FUNCTION_BLOCK CardboardEx EXTENDS SectionEx
VAR_IN_OUT
	benderLeft : FoldingMachine;
	
	robotLeft, robotRight : RobotA22;
	
	skidLeft, skidRight : SkidMagazine;
	magazineLeft, magazineRight : SkidMagazine;
	
	wrapper : WrapMachine;
	
	insertionLeft, insertionRight : Insertion;
	pistonBottom : SimplePiston;
	
	suctionTopLeft : ARRAY[*] OF SuctionPad; (*1..3*)
	suctionTopRight : ARRAY[*] OF SuctionPad; (*1..3*)
	suctionBottomLeft : ARRAY[*] OF SuctionPad; (*1..3*)
	suctionBottomRight : ARRAY[*] OF SuctionPad; (*1..3*)
	
	suctionBottom : ARRAY[*] OF SuctionPad; (*1..2*)
END_VAR
VAR	
	step : (IDLE, LOAD_SIDES_CORNERS, LOAD_TOP_BOTTOM, PUSH, TARGET_WRAP_POSITION, WRAP_AND_RELEASE, COMPLETE := 1050);
	
	masterLoadStep : INT;
	loadStepLeft, loadStepRight : INT;
	
	iWrap : INT;
	wrapPoints : INT;
	wrapRotations : INT;
	masterLength : INT;
	
	releaseDelayTimer : TON;
END_VAR
VAR //local types
	topLeftFoldsArr, topRightFoldsArr, bottomLeftFoldsArr, bottomRightFoldsArr : ARRAY[0..CONSTS.maxPairs] OF INT;
	
	//materialsArr : ARRAY[0..Consts.maxPairs] OF PositionMaterials;
	materialsArr : ARRAY[0..2*Consts.maxPairs] OF PositionMaterials;
	
	recipesCombined : BOOL;
	
	demoHeight : REAL := 640; //mm
	
	innerLoadedMaterials, outerLoadedMaterials : ARRAY[Surface.TOP..Surface.BOTTOM_RIGHT] OF STRING;
	//inner: cardboard by default
	//outer: corner guard by default
END_VAR
VAR CONSTANT
	releaseDelay : TIME := T#2000MS;
END_VAR
VAR
	//AOIs encapsulate functionality and reduce the number of module variables
	aoiCornerGuardLeft, aoiCornerGuardRight : AOI_LoadCornerGuard;
	aoiCornerCardboardLeft, aoiCornerCardboardRight : AOI_LoadCornerCardboard;
	aoiFlatCardboardLeft, aoiFlatCardboardRight : AOI_LoadFlatCardboard;
	
	//for testing only
	latchLeft, latchRight : BOOL; //prevents sliders from overshooting the inner limit sensor
	suctionEnableTopLeft, suctionEnableTopRight, suctionEnableBottomLeft, suctionEnableBottomRight : BOOL;
END_VAR

aoiBlocks();

SUPER^();

METHOD PROTECTED aoiBlocks : BOOL
VAR_INPUT
END_VAR
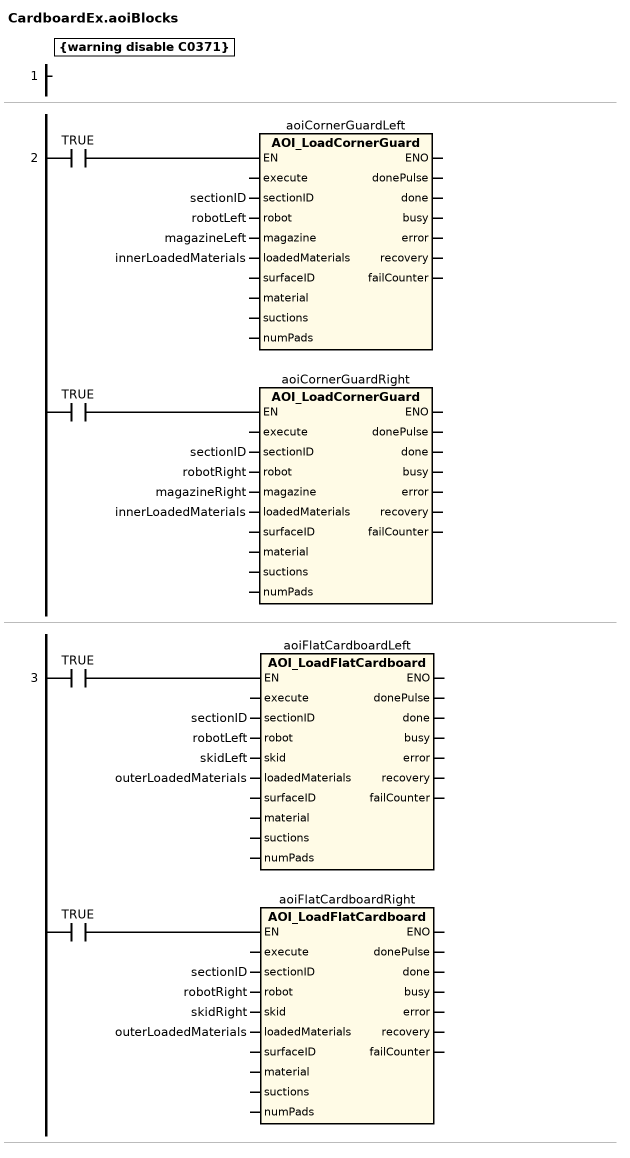
// NETWORK 1
// label: {warning disable C0371}

// NETWORK 2
aoiCornerGuardLeft(
    sectionID := sectionID,
    robot := robotLeft,
    magazine := magazineLeft,
    loadedMaterials := innerLoadedMaterials); // AOI_LoadCornerGuard
aoiCornerGuardRight(
    sectionID := sectionID,
    robot := robotRight,
    magazine := magazineRight,
    loadedMaterials := innerLoadedMaterials); // AOI_LoadCornerGuard

// NETWORK 3
aoiFlatCardboardLeft(
    sectionID := sectionID,
    robot := robotLeft,
    skid := skidLeft,
    loadedMaterials := outerLoadedMaterials); // AOI_LoadFlatCardboard
aoiFlatCardboardRight(
    sectionID := sectionID,
    robot := robotRight,
    skid := skidRight,
    loadedMaterials := outerLoadedMaterials); // AOI_LoadFlatCardboard
END_METHOD

METHOD PROTECTED combine : BOOL
VAR_IN_OUT
	cardboard : ARRAY[*] OF PositionMaterials;
	cornerGuard : ARRAY[*] OF PositionMaterials;
	
	combined : ARRAY[*] OF PositionMaterials;
END_VAR
VAR_INPUT
	cardboard_over_cornerGuard : BOOL;
END_VAR
VAR_INST
	topLength : REAL;
	leftLength : REAL;
	rightLength : REAL;
	bottomLength : REAL;
	
	topLeftLength : REAL;
	topRightLength : REAL;
	bottomLeftLength : REAL;
	bottomRightLength : REAL;
	
	outerMaterialLength : REAL;
	innerMaterialLength : REAL;
	
	i : INT;
	iCardboard : INT;
	iCornerGuard : INT;
END_VAR
FOR i:=0 TO CONSTS.maxPairs*2 BY 1 DO
	IF //no more cardboard (reached end of array or unused entries), 
		(iCardboard >= CONSTS.maxPairs OR_ELSE NOT PositionIsValid(cardboard[iCardboard])) AND_THEN //no more valid cardboard entries
		iCornerGuard < CONSTS.maxPairs AND_THEN //still has remaining corner guard
		PositionIsValid(cornerGuard[iCornerGuard]) //remaining corner guard is valid		
	THEN //finish with cornerguard
		combined[i] := cornerGuard[iCornerGuard];
		iCornerGuard := iCornerGuard + 1;
		CONTINUE;
	END_IF
	
	IF //no more cornerguard (reached end of array or unused entries)
		(iCornerGuard >= CONSTS.maxPairs OR_ELSE NOT PositionIsValid(cornerGuard[iCornerGuard])) AND_THEN
		iCardboard < CONSTS.maxPairs AND_THEN
		PositionIsValid(cardboard[iCardboard])
	THEN //finish with cardboard
		combined[i] := cardboard[iCardboard];
		iCardboard := iCardboard + 1;
		CONTINUE;
	END_IF
	
	(*
	IF NOT cardboard_over_cornerGuard THEN //cardboard on inside
		setOrder(cardboard, cornerGuard, combined, iCardboard, iCornerGuard, i);
		
	ELSE //cardboard on outside
		setOrder(cornerGuard, cardboard, combined, iCornerGuard, iCardboard, i);
		
	END_IF
	*)
END_FOR

combine := TRUE;
END_METHOD

METHOD PROTECTED load : BOOL
VAR_INPUT
	pairIndex : INT;
END_VAR
VAR_OUTPUT
	error : BOOL;
END_VAR
VAR
	pair : REFERENCE TO PositionMaterials REF= materialsArr[pairIndex];
	nextPair : REFERENCE TO PositionMaterials;
END_VAR
(*
unlike other sections, the load() function for cardboard + corner guard only loads the corners
to load flat cardboards, use the function loadFlats()
*)
{warning disable C0371}

IF robotLeft.error OR robotRight.error THEN
	RETURN;
ELSIF NOT (robotLeft.reserve(sectionID) AND robotRight.reserve(sectionID)) THEN //both robots must be reserved first
	RETURN;
END_IF

IF pairIndex + 1 < CONSTS.maxPairs THEN
	nextPair REF= materialsArr[pairIndex + 1];
END_IF

CASE masterLoadStep OF
	0: //check if next pair (which is to be placed over this pair) has the same position as this pair
		IF pairIndex + 1 >= CONSTS.maxPairs THEN //no next pair - NOTE: final pair is index 15 (16-1), not 16
			masterLoadStep := 10;
			loadStepLeft := loadStepRight := 0;
			
		ELSIF pair.position < nextPair.position THEN
			masterLoadStep := 10;
			loadStepLeft := loadStepRight := 0;
		(*	
		ELSIF MatchesMaterialType(pair:= nextPair, materialType:= 'CAR') AND_THEN loadCornerCardboards(pairIndex:= pairIndex + 1) THEN
			masterLoadStep := 10;
			loadStepLeft := loadStepRight := 0;
		*)
		ELSIF MatchesMaterialType(pair:= nextPair, materialPrefix:= 'COR') AND_THEN loadCornerGuards(pairIndex:= pairIndex + 1) THEN
			masterLoadStep := 10;
			loadStepLeft := loadStepRight := 0;
			
		END_IF
		
	10: //load this pair's side cardboards
		IF
			loadFlatCardboardsEx(
				robot:= robotLeft, 
				aoiLoad:= aoiFlatCardboardLeft, 
				loadStep:= loadStepLeft, 
				pairIndex:= pairIndex, 
				includeTop:= FALSE, 
				includeLeft:= TRUE, 
				includeRight:= FALSE, 
				includeBottom:= FALSE, 
				error=> )
			AND
			loadFlatCardboardsEx(
				robot:= robotLeft, 
				aoiLoad:= aoiFlatCardboardLeft, 
				loadStep:= loadStepLeft, 
				pairIndex:= pairIndex, 
				includeTop:= FALSE, 
				includeLeft:= FALSE, 
				includeRight:= TRUE, 
				includeBottom:= FALSE, 
				error=> )
		THEN
			masterLoadStep := 20;
			loadStepLeft := loadStepRight := 0;
		END_IF
		
	20: //load current pair
		IF
			MatchesMaterialType(pair:= pair, materialPrefix:= 'CAR') AND_THEN loadCornerCardboards(pairIndex:= iPair) OR_ELSE
			MatchesMaterialType(pair:= pair, materialPrefix:= 'COR') AND_THEN loadCornerGuards(pairIndex:= iPair)
		THEN //is cardboard
			loadStepLeft := loadStepRight := 0;
			masterLoadStep := COMPLETE;
		END_IF
	
	COMPLETE:
		robotLeft.release(sectionID);
		robotRight.release(sectionID);
		
		loadStepLeft := loadStepRight := 0;
		masterLoadStep := 0;
		load := TRUE;
	
END_CASE
END_METHOD

METHOD PROTECTED loadCornerCardboards : BOOL
VAR_INPUT
	pairIndex : INT;
END_VAR
VAR_OUTPUT
	error : BOOL;
END_VAR
VAR
	errorLeft, errorRight : BOOL;
	leftSuctionArr, rightSuctionArr : POINTER TO SuctionPad;
	leftNextSet, rightNextSet : INT;
	leftMaterial, rightMaterial : STRING;
	leftFold, rightFold : INT;
	
	pair : REFERENCE TO PositionMaterials REF= materialsArr[pairIndex];
	topLeftFold : INT := topLeftFoldsArr[pairIndex];
	topRightFold : INT := topRightFoldsArr[pairIndex];
	bottomLeftFold : INT := bottomLeftFoldsArr[pairIndex];
	bottomRightFold : INT := bottomRightFoldsArr[pairIndex];
END_VAR
{warning disable C0371}

loadCornerCardboards := 
	loadCornerCardboardsEx(
		robot:= robotLeft, 
		aoiLoad:= aoiCornerCardboardLeft, 
		loadStep:= loadStepLeft, 
		pairIndex:= pairIndex, 
		includeTopLeft:= TRUE, 
		includeTopRight:= FALSE, 
		includeBottomLeft:= TRUE, 
		includeBottomRight:= FALSE, 
		error=> errorLeft)
	AND
	loadCornerCardboardsEx(
		robot:= robotRight, 
		aoiLoad:= aoiCornerCardboardRight, 
		loadStep:= loadStepRight, 
		pairIndex:= pairIndex, 
		includeTopLeft:= FALSE, 
		includeTopRight:= TRUE, 
		includeBottomLeft:= FALSE, 
		includeBottomRight:= TRUE, 
		error=> errorLeft);
		
error := errorLeft OR errorRight;

(*
CASE cornerSetLeft OF
	0:
		leftNextSet := Surface.TOP_RIGHT;
		cornerSetLeft := 0;
		
	Surface.TOP_RIGHT: 
		leftNextSet := Surface.TOP_LEFT;
		leftSuctionArr := suctionTopRight;
		leftMaterial := pair.topRight;
		leftFold := topRightFold;
		
	Surface.TOP_LEFT: 
		leftNextSet := Surface.BOTTOM_RIGHT;
		leftSuctionArr := suctionTopLeft;
		leftMaterial := pair.topLeft;
		leftFold := topLeftFold;
		
	Surface.BOTTOM_RIGHT:
		leftNextSet := Surface.BOTTOM_LEFT;
		leftSuctionArr := suctionBottomRight;
		leftMaterial := pair.bottomRight;
		leftFold := bottomRightFold;
		
	Surface.BOTTOM_LEFT: 
		leftNextSet := COMPLETE;
		leftSuctionArr := suctionBottomLeft;
		leftMaterial := pair.bottomLeft;
		leftFold := bottomLeftFold;
END_CASE
IF
	(cornerSetLeft = 0 OR cornerSetLeft = COMPLETE) OR_ELSE
	leftCornerSequence(
		robot:= robotLeft, 
		skid:= skidLeft, 
		suctions := leftSuctionArr,
		loadStep:= loadStepLeft, 
		surfaceID:= cornerSetLeft,
		material:= pair.topRight, 
		foldPos0:= topRightFold, 
		foldPos1:= 0, 
		error=> )
THEN
	cornerSetLeft := leftNextSet;
	loadStepLeft := 0;
END_IF


CASE cornerSetRight OF
	0:
		cornerSetRight := Surface.TOP_RIGHT;
		rightSuctionArr := suctionTopRight;
		
	Surface.TOP_RIGHT:		
		rightNextSet := Surface.BOTTOM_RIGHT;
		rightSuctionArr := suctionTopRight;
		rightMaterial := pair.topRight;
		rightFold := topRightFold;
		
	Surface.BOTTOM_RIGHT: 
		rightNextSet := COMPLETE;
		rightSuctionArr := suctionBottomRight;
		rightMaterial := pair.bottomRight;
		rightFold := bottomRightFold;		
END_CASE
IF
	(cornerSetRight = 0 OR cornerSetRight = COMPLETE) OR_ELSE
	rightCornerSequence(
		robot:= robotRight, 
		skid:= skidRight, 
		suctions := rightSuctionArr,
		loadStep:= loadStepRight, 
		material:= pair.topRight, 
		surfaceID:= cornerSetRight,
		foldPos0:= pair.topRightFold, 
		foldPos1:= 0, 
		error=> )
THEN
	cornerSetRight := rightNextSet;
	loadStepRight := 0;
END_IF



IF cornerSetLeft = COMPLETE AND cornerSetRight = COMPLETE THEN
	loadCornerCardboards := TRUE;
	
	loadStepLeft := loadStepRight := 0;
	cornerSetLeft := cornerSetRight := 0;
END_IF
*)
END_METHOD

METHOD PROTECTED loadCornerCardboardsEx : BOOL
VAR_IN_OUT
	robot : RobotA22;
	aoiLoad : AOI_LoadCornerCardboard;
	loadStep : INT;
END_VAR
VAR_INPUT
	pairIndex : INT;
	includeTopLeft, includeTopRight, includeBottomLeft, includeBottomRight : BOOL;
END_VAR
VAR_OUTPUT
	error : BOOL;
END_VAR
VAR
	suctionsArrLeft, suctionsArrRight : POINTER TO SuctionPad;
	nextSetLeft, nextSetRight : INT;

	pair : REFERENCE TO PositionMaterials REF= materialsArr[pairIndex];
	topLeftFold : INT := topLeftFoldsArr[pairIndex];
	topRightFold : INT := topRightFoldsArr[pairIndex];
	bottomLeftFold : INT := bottomLeftFoldsArr[pairIndex];
	bottomRightFold : INT := bottomRightFoldsArr[pairIndex];
END_VAR
{warning disable C0371}

IF robot.error THEN
	error := TRUE;
	RETURN;
ELSIF robot.reservation <> sectionID AND_THEN NOT robot.reserve(sectionID) THEN
	RETURN;
ELSIF robot.tool <> sectionID AND_THEN NOT robot.changeEOAT(targetTool := sectionID) THEN
	RETURN;
END_IF

error := aoiLoad.error;

CASE loadStep OF
	0:
		loadStep := Surface.BOTTOM_LEFT;
		
	Surface.BOTTOM_LEFT:
		IF NOT includeBottomLeft OR aoiLoad.donePulse THEN
			aoiLoad.execute := FALSE;
			aoiLoad.material := '';
			loadStep := Surface.BOTTOM_RIGHT;
			RETURN;
		END_IF
		
		aoiLoad.surfaceID := loadStep;
		aoiLoad.material := pair.bottomLeft;
		aoiLoad.suctions := suctionBottomLeft;
		aoiLoad.numPads := UPPER_BOUND(suctionBottomLeft, 1) - LOWER_BOUND(suctionBottomLeft, 1) + 1;
		
		aoiLoad.foldPos0 := bottomLeftFold;
		aoiLoad.foldPos1 := 0;
		
		aoiLoad.execute := NOT aoiLoad.busy;
		
	Surface.BOTTOM_RIGHT:
		IF NOT includeBottomRight OR aoiLoad.donePulse THEN
			aoiLoad.execute := FALSE;
			aoiLoad.material := '';
			loadStep := Surface.TOP_LEFT;
			RETURN;
		END_IF
		
		aoiLoad.surfaceID := loadStep;
		aoiLoad.material := pair.bottomRight;
		aoiLoad.suctions := suctionBottomRight;
		aoiLoad.numPads := UPPER_BOUND(suctionBottomRight, 1) - LOWER_BOUND(suctionBottomRight, 1) + 1;
		
		aoiLoad.foldPos0 := bottomRightFold;
		aoiLoad.foldPos1 := 0;
		
		aoiLoad.execute := NOT aoiLoad.busy;
	
	Surface.TOP_LEFT:		
		IF NOT includeTopLeft OR aoiLoad.donePulse THEN
			aoiLoad.execute := FALSE;
			aoiLoad.material := '';
			loadStep := Surface.TOP_RIGHT;
			RETURN;
		END_IF
		
		aoiLoad.surfaceID := loadStep;
		aoiLoad.material := pair.top;
		aoiLoad.suctions := suctionTopLeft;
		aoiLoad.numPads := UPPER_BOUND(suctionTopLeft, 1) - LOWER_BOUND(suctionTopLeft, 1) + 1;
		
		aoiLoad.foldPos0 := topLeftFold;
		aoiLoad.foldPos1 := 0;
		
		aoiLoad.execute := NOT aoiLoad.busy;
		
	Surface.TOP_RIGHT:
		IF NOT includeTopRight OR aoiLoad.donePulse THEN
			aoiLoad.execute := FALSE;
			aoiLoad.material := '';
			loadStep := COMPLETE;
			RETURN;
		END_IF
		
		aoiLoad.surfaceID := loadStep;
		aoiLoad.material := pair.topRight;
		aoiLoad.suctions := suctionTopRight;
		aoiLoad.numPads := UPPER_BOUND(suctionTopRight, 1) - LOWER_BOUND(suctionTopRight, 1) + 1;
		
		aoiLoad.foldPos0 := topRightFold;
		aoiLoad.foldPos1 := 0;
		
		aoiLoad.execute := NOT aoiLoad.busy;
		
	COMPLETE:				
		robot.release(sectionID);
		
		aoiLoad.material := '';
		aoiLoad.execute := FALSE;
		
		loadCornerCardboardsEx := TRUE;
END_CASE
END_METHOD

METHOD loadCornerGuards : BOOL
VAR_INPUT
	pairIndex : INT;
END_VAR
VAR_OUTPUT
	error : BOOL;
END_VAR
VAR
	pair : REFERENCE TO PositionMaterials REF= materialsArr[pairIndex];
	errorLeft, errorRight : BOOL;
END_VAR
{warning disable C0371}

loadCornerGuards := 
	loadCornerGuardsEx(
		robot:= robotLeft, 
		aoiLoad:= aoiCornerGuardLeft, 
		loadStep:= loadStepLeft, 
		pairIndex:= pairIndex, 
		includeTopLeft:= TRUE, 
		includeTopRight:= FALSE, 
		includeBottomLeft:= TRUE, 
		includeBottomRight:= FALSE, 
		error=> errorLeft) 
	AND
	loadCornerGuardsEx(
		robot:= robotRight, 
		aoiLoad:= aoiCornerGuardRight, 
		loadStep:= loadStepRight, 
		pairIndex:= pairIndex, 
		includeTopLeft:= FALSE, 
		includeTopRight:= TRUE, 
		includeBottomLeft:= FALSE, 
		includeBottomRight:= TRUE, 
		error=> errorRight);
		
error := errorLeft OR errorRight;

(*
IF robotLeft.error OR robotRight.error THEN
	error := TRUE;
	RETURN;
	
ELSIF 
	(robotLeft.reservation <> sectionID AND_THEN NOT robotLeft.reserve(sectionID)) OR 
	(robotRight.reservation <> sectionID AND_THEN NOT robotRight.reserve(sectionID))
THEN //loading requires both robots be reserved together
	RETURN;
	
ELSIF //robots have wrong tool
	(robotLeft.tool <> sectionID AND_THEN NOT robotLeft.changeEOAT(targetTool := sectionID)) OR
	(robotRight.tool <> sectionID AND_THEN NOT robotRight.changeEOAT(targetTool := sectionID))
THEN
	RETURN;
	
END_IF

CASE loadStep OF
	0: //top and bottom
		IF aoiCornerGuardLeft.done AND aoiCornerGuardRight.done THEN
			aoiCornerGuardLeft.execute := aoiCornerGuardRight.execute := FALSE;
			aoiCornerGuardLeft.material := aoiCornerGuardRight.material := '';
			loadStep := 10;
			RETURN;
		END_IF
		
		aoiCornerGuardLeft.suctions := 0;
		aoiCornerGuardLeft.surfaceID := Surface.TOP;
		aoiCornerGuardLeft.material := pair.top;
		aoiCornerGuardLeft.numPads := 0;
		
		aoiCornerGuardRight.suctions := suctionBottom;
		aoiCornerGuardRight.surfaceID := Surface.BOTTOM;
		aoiCornerGuardRight.material := pair.bottom;
		aoiCornerGuardRight.numPads := 0;
		
		aoiCornerGuardLeft.execute := NOT aoiCornerGuardLeft.done AND NOT aoiCornerGuardLeft.busy;
		aoiCornerGuardRight.execute := NOT aoiCornerGuardRight.done AND NOT aoiCornerGuardRight.busy;
		
	10: //sides
		IF aoiCornerGuardLeft.done AND aoiCornerGuardRight.done THEN
			aoiCornerGuardLeft.execute := aoiCornerGuardRight.execute := FALSE;
			aoiCornerGuardLeft.material := aoiCornerGuardRight.material := '';
			loadStep := 10;
			RETURN;
		END_IF
		
		aoiCornerGuardLeft.suctions := 0;
		aoiCornerGuardLeft.surfaceID := Surface.LEFT;
		aoiCornerGuardLeft.material := pair.left;
		aoiCornerGuardLeft.numPads := 0;
		
		aoiCornerGuardRight.suctions := 0;
		aoiCornerGuardRight.surfaceID := Surface.RIGHT;
		aoiCornerGuardRight.material := pair.right;
		aoiCornerGuardRight.numPads := 0;
		
		aoiCornerGuardLeft.execute := NOT aoiCornerGuardLeft.done AND NOT aoiCornerGuardLeft.busy;
		aoiCornerGuardRight.execute := NOT aoiCornerGuardRight.done AND NOT aoiCornerGuardRight.busy;
		
	COMPLETE:
		loadStep := 0;
		loadCornerGuards := TRUE;
END_CASE

error := aoiCornerGuardLeft.error OR aoiCornerGuardRight.error;
*)
END_METHOD

METHOD loadCornerGuardsEx : BOOL
VAR_IN_OUT
	robot : RobotA22;
	aoiLoad : AOI_LoadCornerGuard;
	loadStep : INT;
END_VAR
VAR_INPUT
	pairIndex : INT;
	includeTopLeft, includeTopRight, includeBottomLeft, includeBottomRight : BOOL;
END_VAR
VAR_OUTPUT
	error : BOOL;
END_VAR
VAR
	pair : REFERENCE TO PositionMaterials REF= materialsArr[pairIndex];
END_VAR
{warning disable C0371}
IF robot.error THEN
	error := TRUE;
	RETURN;
ELSIF robot.reservation <> sectionID AND_THEN NOT robot.reserve(sectionID) THEN
	RETURN;
ELSIF robot.tool <> sectionID AND_THEN NOT robot.changeEOAT(targetTool := sectionID) THEN
	RETURN;
END_IF

error := aoiLoad.error;

CASE loadStep OF
	0:
		loadStep := Surface.BOTTOM_LEFT;
		
	Surface.BOTTOM_LEFT:
		IF NOT includeBottomLeft OR aoiLoad.donePulse THEN
			aoiLoad.execute := FALSE;
			aoiLoad.material := '';
			loadStep := Surface.BOTTOM_RIGHT;
			RETURN;
		END_IF
		
		aoiLoad.surfaceID := loadStep;
		aoiLoad.material := pair.bottomLeft;
		aoiLoad.suctions := suctionBottomLeft;
		aoiLoad.numPads := UPPER_BOUND(suctionBottomLeft, 1) - LOWER_BOUND(suctionBottomLeft, 1) + 1;
		
		aoiLoad.execute := NOT aoiLoad.busy;
		
	Surface.BOTTOM_RIGHT:
		IF NOT includeBottomRight OR aoiLoad.donePulse THEN
			aoiLoad.execute := FALSE;
			aoiLoad.material := '';
			loadStep := Surface.TOP_LEFT;
			RETURN;
		END_IF
		
		aoiLoad.surfaceID := loadStep;
		aoiLoad.material := pair.bottomRight;
		aoiLoad.suctions := suctionBottomRight;
		aoiLoad.numPads := UPPER_BOUND(suctionBottomRight, 1) - LOWER_BOUND(suctionBottomRight, 1) + 1;
		
		aoiLoad.execute := NOT aoiLoad.busy;
	
	Surface.TOP_LEFT:		
		IF NOT includeTopLeft OR aoiLoad.donePulse THEN
			aoiLoad.execute := FALSE;
			aoiLoad.material := '';
			loadStep := Surface.TOP_RIGHT;
			RETURN;
		END_IF
		
		aoiLoad.surfaceID := loadStep;
		aoiLoad.material := pair.top;
		aoiLoad.suctions := suctionTopLeft;
		aoiLoad.numPads := UPPER_BOUND(suctionTopLeft, 1) - LOWER_BOUND(suctionTopLeft, 1) + 1;
		
		aoiLoad.execute := NOT aoiLoad.busy;
		
	Surface.TOP_RIGHT:
		IF NOT includeTopRight OR aoiLoad.donePulse THEN
			aoiLoad.execute := FALSE;
			aoiLoad.material := '';
			loadStep := COMPLETE;
			RETURN;
		END_IF
		
		aoiLoad.surfaceID := loadStep;
		aoiLoad.material := pair.topRight;
		aoiLoad.suctions := suctionTopRight;
		aoiLoad.numPads := UPPER_BOUND(suctionTopRight, 1) - LOWER_BOUND(suctionTopRight, 1) + 1;
		
		aoiLoad.execute := NOT aoiLoad.busy;
		
	COMPLETE:				
		robot.release(sectionID);
		
		aoiLoad.material := '';
		aoiLoad.execute := FALSE;
		
		loadCornerGuardsEx := TRUE;
END_CASE
END_METHOD

METHOD PROTECTED loadFlatCardboards : BOOL
VAR_INPUT
	pairIndex : INT;
END_VAR
VAR_OUTPUT
	error : BOOL;
END_VAR
VAR
	pair : REFERENCE TO PositionMaterials REF= materialsArr[pairIndex];
	errorLeft, errorRight : BOOL;
END_VAR
{warning disable C0371}

loadFlatCardboards := 
	loadFlatCardboardsEx(
		robot:= robotLeft, 
		aoiLoad:= aoiFlatCardboardLeft, 
		loadStep:= loadStepLeft, 
		pairIndex:= pairIndex, 
		includeTop:= TRUE, 
		includeLeft:= FALSE, //left already loaded before
		includeRight:= FALSE, 
		includeBottom:= FALSE, 
		error=> errorLeft)
	AND
	loadFlatCardboardsEx(
		robot:= robotRight, 
		aoiLoad:= aoiFlatCardboardRight, 
		loadStep:= loadStepRight, 
		pairIndex:= pairIndex, 
		includeTop:= FALSE, 
		includeLeft:= FALSE, 
		includeRight:= FALSE, //right already loaded before
		includeBottom:= TRUE, 
		error=> errorRight);
		
error := errorLeft OR errorRight;

(*
IF robotLeft.error OR robotRight.error THEN
	error := TRUE;
	RETURN;
	
ELSIF 
	(robotLeft.reservation <> sectionID AND_THEN NOT robotLeft.reserve(sectionID)) OR 
	(robotRight.reservation <> sectionID AND_THEN NOT robotRight.reserve(sectionID))
THEN //loading requires both robots be reserved together
	RETURN;
	
ELSIF //robots have wrong tool
	(robotLeft.tool <> sectionID AND_THEN NOT robotLeft.changeEOAT(targetTool := sectionID)) OR
	(robotRight.tool <> sectionID AND_THEN NOT robotRight.changeEOAT(targetTool := sectionID))
THEN
	RETURN;
	
END_IF

CASE loadStep OF
	0: //top and bottom
		IF aoiFlatCardboardLeft.done AND aoiFlatCardboardRight.done THEN
			aoiFlatCardboardLeft.execute := aoiFlatCardboardRight.execute := FALSE;
			aoiFlatCardboardLeft.material := aoiFlatCardboardRight.material := '';
			loadStep := 10;
			RETURN;
		END_IF
		
		aoiFlatCardboardLeft.suctions := 0;
		aoiFlatCardboardLeft.surfaceID := Surface.TOP;
		aoiFlatCardboardLeft.material := pair.top;
		aoiFlatCardboardLeft.numPads := 0;
		
		aoiFlatCardboardRight.suctions := suctionBottom;
		aoiFlatCardboardRight.surfaceID := Surface.BOTTOM;
		aoiFlatCardboardRight.material := pair.bottom;
		aoiFlatCardboardRight.numPads := 0;
		
		aoiFlatCardboardLeft.execute := NOT aoiFlatCardboardLeft.done AND NOT aoiFlatCardboardLeft.busy;
		aoiFlatCardboardRight.execute := NOT aoiFlatCardboardRight.done AND NOT aoiFlatCardboardRight.busy;
		
	10: //sides
		IF aoiFlatCardboardLeft.done AND aoiFlatCardboardRight.done THEN
			aoiFlatCardboardLeft.execute := aoiFlatCardboardRight.execute := FALSE;
			aoiFlatCardboardLeft.material := aoiFlatCardboardRight.material := '';
			loadStep := 10;
			RETURN;
		END_IF
		
		aoiFlatCardboardLeft.suctions := 0;
		aoiFlatCardboardLeft.surfaceID := Surface.LEFT;
		aoiFlatCardboardLeft.material := pair.left;
		aoiFlatCardboardLeft.numPads := 0;
		
		aoiFlatCardboardRight.suctions := 0;
		aoiFlatCardboardRight.surfaceID := Surface.RIGHT;
		aoiFlatCardboardRight.material := pair.right;
		aoiFlatCardboardRight.numPads := 0;
		
		aoiFlatCardboardLeft.execute := NOT aoiFlatCardboardLeft.done AND NOT aoiFlatCardboardLeft.busy;
		aoiFlatCardboardRight.execute := NOT aoiFlatCardboardRight.done AND NOT aoiFlatCardboardRight.busy;
		
	COMPLETE:
		loadStepLeft := loadStepRight := 0;
		loadStep := 0;
		
		loadFlatCardboards := TRUE;
END_CASE

error := aoiFlatCardboardLeft.error OR aoiFlatCardboardRight.error;
*)
END_METHOD

METHOD loadFlatCardboardsEx : BOOL
VAR_IN_OUT
	robot : RobotA22;
	aoiLoad : AOI_LoadFlatCardboard;
	loadStep : INT;
END_VAR
VAR_INPUT
	pairIndex : INT;
	includeTop, includeLeft, includeRight, includeBottom : BOOL;
END_VAR
VAR_OUTPUT
	error : BOOL;
END_VAR
VAR
	pair : REFERENCE TO PositionMaterials REF= materialsArr[pairIndex];
END_VAR
IF robot.error THEN
	error := TRUE;
	RETURN;
ELSIF robot.reservation <> sectionID AND_THEN NOT robot.reserve(sectionID) THEN
	RETURN;
ELSIF robot.tool <> sectionID AND_THEN NOT robot.changeEOAT(targetTool := sectionID) THEN
	RETURN;
END_IF

error := aoiLoad.error;

CASE loadStep OF
	0:
		loadStep := Surface.TOP;
	
	Surface.TOP:	
		IF NOT includeTop OR aoiLoad.donePulse THEN
			aoiLoad.execute := FALSE;
			aoiLoad.material := '';
			loadStep := Surface.BOTTOM;
			RETURN;
		END_IF
		
		aoiLoad.surfaceID := Surface.TOP;
		aoiLoad.material := pair.top;
		aoiLoad.suctions := 0;
		aoiLoad.numPads := 0;
		
		aoiLoad.execute := NOT aoiLoad.busy;
		
	Surface.BOTTOM:
		IF NOT includeBottom OR aoiLoad.donePulse THEN
			aoiLoad.execute := FALSE;
			aoiLoad.material := '';
			loadStep := Surface.LEFT;
			RETURN;
		END_IF
		
		aoiLoad.surfaceID := Surface.BOTTOM;
		aoiLoad.material := pair.bottom;
		aoiLoad.suctions := suctionBottom;
		aoiLoad.numPads := UPPER_BOUND(suctionBottom, 1) - LOWER_BOUND(suctionBottom, 1) + 1;
		
		aoiLoad.execute := NOT aoiLoad.busy;
		
	Surface.LEFT:
		IF NOT includeLeft OR aoiLoad.donePulse THEN
			aoiLoad.execute := FALSE;
			aoiLoad.material := '';
			loadStep := Surface.RIGHT;
			RETURN;
		END_IF
		
		aoiLoad.surfaceID := Surface.LEFT;
		aoiLoad.material := pair.left;
		aoiLoad.suctions := 0;
		aoiLoad.numPads := 0;
		
		aoiLoad.execute := NOT aoiLoad.busy;
		
	Surface.RIGHT:
		IF NOT includeRight OR aoiLoad.donePulse THEN
			aoiLoad.execute := FALSE;
			aoiLoad.material := '';
			loadStep := COMPLETE;
			RETURN;
		END_IF
		
		aoiLoad.surfaceID := Surface.RIGHT;
		aoiLoad.material := pair.right;
		aoiLoad.suctions := 0;
		aoiLoad.numPads := 0;
		
		aoiLoad.execute := NOT aoiLoad.busy;
		
	COMPLETE:				
		robot.release(sectionID);
		
		aoiLoad.material := '';
		aoiLoad.execute := FALSE;
		
		loadFlatCardboardsEx := TRUE;
END_CASE
END_METHOD

METHOD PROTECTED maintenance : BOOL
VAR_INPUT
END_VAR
{warning disable C0371}
IF robotLeft.Done THEN
	robotLeft.clearCommand();
END_IF

IF robotRight.Done THEN
	robotRight.clearCommand();
END_IF
END_METHOD

METHOD PROTECTED manual : BOOL
VAR_INPUT
END_VAR
END_METHOD

METHOD PROTECTED process : BOOL
VAR_INPUT
	auto : BOOL;
END_VAR
VAR_OUTPUT
	error : BOOL;
END_VAR
VAR
	currentPair : REFERENCE TO PositionMaterials REF= materialsArr[iPair];
END_VAR
{warning disable C0371}

IF iPair >= CONSTS.maxPairs THEN
	process := TRUE;
	RETURN;
ELSIF NOT PositionIsValid(pair := currentPair) THEN
	iPair := iPair + 1;
	RETURN;
END_IF
(*
corrected sequence:
	load sides
	load corners
	load bottom
	load top
*)

CASE step OF
	IDLE:
		IF trigger.Q THEN
			step := LOAD_SIDES_CORNERS;
		END_IF
	
	LOAD_SIDES_CORNERS: //load
		IF
			(auto AND done) OR
			(NOT auto AND trigger.Q)
		THEN
			aoiCornerCardboardLeft.reset();
			aoiCornerCardboardRight.reset();
			
			aoiCornerGuardLeft.reset();
			aoiCornerGuardRight.reset();
			
			aoiFlatCardboardLeft.reset();
			aoiFlatCardboardRight.reset();
			
			step := LOAD_TOP_BOTTOM;
			RETURN;
		END_IF
		
		IF NOT done THEN
			done := load(pairIndex := iPair);
		END_IF
		
	LOAD_TOP_BOTTOM:
		IF
			(auto AND done) OR
			(NOT auto AND trigger.Q)
		THEN
			aoiCornerCardboardLeft.reset();
			aoiCornerCardboardRight.reset();
			
			aoiCornerGuardLeft.reset();
			aoiCornerGuardRight.reset();
			
			aoiFlatCardboardLeft.reset();
			aoiFlatCardboardRight.reset();
			
			step := PUSH;
			RETURN;
		END_IF
		
		IF NOT done THEN
			done := loadFlatCardboards(pairIndex := iPair);
		END_IF
		
	PUSH:
		IF
			(auto AND latchLeft AND latchRight AND pistonBottom.extended) OR
			(NOT auto AND trigger.Q)
		THEN
			step := TARGET_WRAP_POSITION;
			RETURN;
		END_IF
		
		insertionLeft.align(demoHeight+5);
		insertionRight.align(demoHeight+5);
		
		IF //align slider to 5mm gap above bundle height
			insertionLeft.sliderPos <> demoHeight+5 OR
			insertionRight.sliderPos <> demoHeight+5
		THEN
			RETURN;
		END_IF
		
		IF NOT latchLeft THEN
			latchLeft := insertionLeft.contact;
			insertionLeft.press();
		END_IF
		
		IF NOT latchRight THEN
			latchRight := insertionRight.contact;
			insertionRight.press();
		END_IF
		
		pistonBottom.extend();
		
	TARGET_WRAP_POSITION:		
		IF iWrap >= wrapPoints THEN
			step := COMPLETE;
			RETURN;
		END_IF
		
		IF materialsArr[iPair].position = materialsArr[iPair + 1].position THEN //if this and the next pair were loaded together
			masterLength := TO_INT( MAX( GetPairMasterLength(materialsArr[iPair]), GetPairMasterLength(materialsArr[iPair + 1]) ) );
			wrapPoints := MAX( materialsArr[iPair].wrapPoints, materialsArr[iPair + 1].wrapPoints );
			wrapRotations := MAX( materialsArr[iPair].wrapRotations, materialsArr[iPair + 1].wrapRotations );
		ELSE
			masterLength := TO_INT( GetPairMasterLength(materialsArr[iPair]) );
			wrapPoints := materialsArr[iPair].wrapPoints;
			wrapRotations := materialsArr[iPair].wrapRotations;
		END_IF
		
		(*
		directionCheckAndSet(
			wrapConveyorPos,
			(currentPair.position - masterLength/2) + (masterLength/(currentPair.wrapPoints + 1) * (iWrap + 1)));
		*)
		step := WRAP_AND_RELEASE;
		
	WRAP_AND_RELEASE:
		releaseDelayTimer(IN:= , PT:= releaseDelay, Q=> , ET=> );
		
		IF wrapper.ready THEN
			wrapper.wrap(wrapRotations);
			releaseDelayTimer.IN := TRUE;
		END_IF
		
		IF releaseDelayTimer.Q THEN
			SetSuctions(suctions := suctionTopLeft, state := FALSE);
			SetSuctions(suctions := suctionTopRight, state := FALSE);
			SetSuctions(suctions := suctionBottomLeft, state := FALSE);
			SetSuctions(suctions := suctionBottomRight, state := FALSE);
			
			insertionLeft.toHome();
			insertionRight.toHome();
			pistonBottom.retract();
		END_IF
		
		IF wrapper.done AND insertionLeft.home AND insertionRight.home AND pistonBottom.retracted THEN
			releaseDelayTimer.IN := FALSE;
			step := WRAP_AND_RELEASE;
		END_IF
	
	COMPLETE:
		iPair := iPair + 1;
		iWrap := wrapPoints := wrapRotations := 0;
		step := IDLE;
		
END_CASE
END_METHOD

METHOD PROTECTED ps_AbortCondition : BOOL
VAR_INPUT
END_VAR
{warning disable C0371}
ps_AbortCondition :=
	insertionLeft.error OR 
	insertionRight.error OR 
	robotLeft.error OR 
	robotRight.error OR
	wrapper.error;
END_METHOD

METHOD PROTECTED ps_Aborted : BOOL
VAR_INPUT
END_VAR
ps_Aborted := TRUE;
END_METHOD

METHOD PROTECTED ps_Aborting : BOOL
VAR_INPUT
END_VAR
{warning disable C0371}
insertionLeft.stop();
insertionRight.stop();
pistonBottom.stop();

aoiFlatCardboardLeft.reset();
aoiFlatCardboardRight.reset();

aoiCornerCardboardLeft.reset();
aoiCornerCardboardRight.reset();

aoiCornerGuardLeft.reset();
aoiCornerGuardRight.reset();

robotLeft.clearCommand();
robotRight.clearCommand();

//stop conveyors

ps_Aborting :=
	NOT insertionLeft.active AND
	NOT insertionRight.active AND
	NOT pistonBottom.busy AND
	NOT robotLeft.Busy AND
	NOT robotRight.Busy;
END_METHOD

METHOD PROTECTED ps_Clearing : BOOL
VAR_INPUT
END_VAR
{warning disable C0371}
insertionLeft.reset();
insertionRight.reset();

ps_Clearing := 
	NOT insertionLeft.error AND
	NOT insertionRight.error AND
	NOT wrapper.error AND
	NOT robotLeft.error AND
	NOT robotRight.error;
END_METHOD

METHOD PROTECTED ps_Complete : BOOL
VAR_INPUT
END_VAR
ps_Complete := TRUE;
END_METHOD

METHOD PROTECTED ps_Completing : BOOL
VAR_INPUT
END_VAR
ps_Completing := NOT occupied;
END_METHOD

METHOD PROTECTED ps_Held : BOOL
VAR_INPUT
END_VAR
ps_Held := NOT hold;
END_METHOD

METHOD PROTECTED ps_HoldCondition : BOOL
VAR_INPUT
END_VAR
END_METHOD

METHOD PROTECTED ps_Holding : BOOL
VAR_INPUT
END_VAR
{warning disable C0371}
insertionLeft.stop();
insertionRight.stop();
pistonBottom.stop();
//set robot to pause

ps_Holding :=
	NOT insertionLeft.active AND
	NOT insertionRight.active;
END_METHOD

METHOD PROTECTED ps_Resetting : BOOL
VAR_INPUT
END_VAR
{warning disable C0371}
insertionLeft.reset();
insertionRight.reset();

ps_Resetting := 
	reset AND
	NOT insertionLeft.error AND
	NOT insertionRight.error AND
	NOT wrapper.error AND
	NOT robotLeft.error AND
	NOT robotRight.error;
END_METHOD

METHOD PROTECTED ps_Starting : BOOL
VAR_INPUT
END_VAR
{warning disable C0371}
robotLeft.clearCommand();
robotRight.clearCommand();

insertionLeft.homingSequence();
insertionRight.homingSequence();
pistonBottom.retract();

ps_Starting := 
	insertionLeft.screw.HomeSet AND 
	insertionRight.screw.HomeSet AND 
	pistonBottom.retracted;
END_METHOD

METHOD PROTECTED ps_StopCondition : BOOL
VAR_INPUT
END_VAR
ps_StopCondition := 
	stop;
END_METHOD

METHOD PROTECTED ps_Stopped : BOOL
VAR_INPUT
END_VAR
ps_Stopped := TRUE;
END_METHOD

METHOD PROTECTED ps_Stopping : BOOL
VAR_INPUT
END_VAR
{warning disable C0371}
insertionLeft.stop();
insertionRight.stop();
pistonBottom.stop();

aoiFlatCardboardLeft.reset();
aoiFlatCardboardRight.reset();

aoiCornerCardboardLeft.reset();
aoiCornerCardboardRight.reset();

aoiCornerGuardLeft.reset();
aoiCornerGuardRight.reset();

robotLeft.clearCommand();
robotRight.clearCommand();

wrapper.bEnable := FALSE;

//stop conveyors

ps_Stopping :=
	//NOT insertionLeft.active AND
	NOT insertionRight.active AND
	NOT pistonBottom.busy AND
	NOT robotLeft.Busy AND
	NOT robotRight.Busy AND
	NOT wrapper.busy;
END_METHOD

METHOD PROTECTED ps_SuspendCondition : BOOL
VAR_INPUT
END_VAR
END_METHOD

METHOD PROTECTED ps_Suspended : BOOL
VAR_INPUT
END_VAR
ps_Suspended := NOT ps_SuspendCondition();
END_METHOD

METHOD PROTECTED ps_Suspending : BOOL
VAR_INPUT
END_VAR
ps_Suspending := TRUE;
END_METHOD

METHOD PROTECTED ps_Unholding : BOOL
VAR_INPUT
END_VAR
ps_Unholding := TRUE;
END_METHOD

METHOD PROTECTED ps_Unsuspending : BOOL
VAR_INPUT
END_VAR
ps_Unsuspending := TRUE;
END_METHOD

METHOD PROTECTED runSectionTasks : BOOL
VAR_INPUT
	auto : BOOL;
END_VAR
VAR_OUTPUT
	error : BOOL;
END_VAR
SUPER^.runSectionTasks(auto := auto, error => error);

CASE status OF
	SectionTask.IDLE:
		RETURN;
	
	SectionTask.ALIGN:
		IF NOT recipesCombined THEN
			combine(
				currentBundle.cardboard, 
				currentBundle.cornerGuard, 
				materialsArr, 
				currentBundle.cardboard_over_cornerGuard);
				
			recipesCombined := TRUE;
		END_IF
		
	SectionTask.ACTIVE:
		recipesCombined := FALSE;
		
	SectionTask.DISCHARGE:
		//
		
	SectionTask.COMPLETE:	
		//
		
	-100:
		RETURN;
		
END_CASE
END_METHOD

METHOD PROTECTED setOrder : BOOL
VAR_IN_OUT
	innerArray : ARRAY[*] OF PositionMaterials;
	outerArray : ARRAY[*] OF PositionMaterials;
	
	combined : ARRAY[*] OF PositionMaterials;
	
	i_inner : INT;
	i_outer : INT;
	i_combined : INT;
END_VAR
VAR	
	outerMaterialLength : LREAL;
	innerMaterialLength : LREAL;
END_VAR
//if inner material is in front of outer material, inner material goes first
IF innerArray[i_inner].position <= outerArray[i_outer].position THEN

	combined[i_combined] := innerArray[i_inner];
	i_inner := i_inner + 1; //check next cardboard during next iteration
	
	setOrder := TRUE;
	RETURN;
END_IF
	
outerMaterialLength := GetPairMasterLength(outerArray[i_outer]);
innerMaterialLength := GetPairMasterLength(innerArray[i_inner]);

//if current inner material is too close to current outer material, place inner material first
//compare inner materials' front with outer material's back
IF (innerArray[i_inner].position - innerMaterialLength/2) < (outerArray[i_outer].position + outerMaterialLength/2) THEN
	combined[i_combined] := innerArray[i_inner];
	i_inner := i_inner + 1;
ELSE //otherwise, outer material can go
	combined[i_combined] := outerArray[i_outer];
	i_outer := i_outer + 1;
END_IF

setOrder := TRUE;
END_METHOD

METHOD PROTECTED unload : BOOL
VAR_INPUT
END_VAR
END_METHOD

END_FUNCTION_BLOCK

(* stored: Version 1.1.0.1, ProductVersion 3.1.4024.11
   POU CardboardEx: Id {43a9c6e1-e77d-41f5-aea3-07b47a57c140}, SpecialFunc None
   Folder Actions_Cyclic: Id {c8c39f76-dbed-4e64-98b8-9f897e55ef48}
   Folder Corner Cardboard: Id {ae97f731-8159-458d-a4c2-1a1c4ac5d0d1}
   Folder Corner Guards: Id {1633509f-8083-40cb-8029-83f401dfca46}
   Folder Flat Cardboard: Id {ccd7d2aa-e76b-439c-81f7-22b0db1787fb}
   Folder PML Conditions: Id {59aefde4-737b-476f-91c3-16f03e5b5428}
   Folder PML Inter. States: Id {209a759f-9928-4b87-9e7f-059f48bd90b9}
   Folder Recipe Combination: Id {e84711e1-12c7-48bc-a0fc-ee5336e88119}
   Method aoiBlocks: Id {e19d7a5d-07d7-472d-bc72-4c28bb47c7dc}
   Method combine: Id {68c0a6ae-b842-4781-b6e7-e5f46d476b9d}
   Method load: Id {a681c93d-e590-4020-9185-d7ae010cf638}
   Method loadCornerCardboards: Id {fc6e26f1-7233-42c4-a94a-66d2e256266a}
   Method loadCornerCardboardsEx: Id {156f628d-7b56-4840-9717-9971eeb42365}
   Method loadCornerGuards: Id {f8d7145e-2601-4096-b20d-bfa97c3f5492}
   Method loadCornerGuardsEx: Id {ac43d9ca-0f0f-4142-b559-dd30cf7e65a4}
   Method loadFlatCardboards: Id {b9a93d4c-938b-4af6-a5a3-5141d50c48d4}
   Method loadFlatCardboardsEx: Id {a6006f45-57d8-4c80-8e03-0111060a1c4e}
   Method maintenance: Id {8dc492fc-7c74-48c6-a0e8-0f621ee44eb4}
   Method manual: Id {27f7e290-328e-4f21-8768-c59937f9f3f4}
   Method process: Id {12873255-c3e6-4f5b-bcd2-07be3d909921}
   Method ps_AbortCondition: Id {9a23cbff-07db-45fb-bc55-9ee98df4fcd2}
   Method ps_Aborted: Id {29be6b49-0b62-4a69-87e2-c759f383d316}
   Method ps_Aborting: Id {b2ad3988-d8ea-4219-bf7d-f35e1a9ed0f7}
   Method ps_Clearing: Id {91f61558-4792-4680-a9c0-e278e2be45e2}
   Method ps_Complete: Id {9630f40f-1ae3-4300-8f07-f6ffb8ca5dcd}
   Method ps_Completing: Id {e9302788-bb7d-4882-8053-556af19fbbd7}
   Method ps_Held: Id {5952d544-ae8a-4198-afb3-ad748cffd145}
   Method ps_HoldCondition: Id {db7a9fa0-a521-4806-a018-ed7babca466e}
   Method ps_Holding: Id {25454e92-6403-48af-afec-3a7ce519f1f2}
   Method ps_Resetting: Id {161cd2ee-cfcf-492e-bbdb-d07619fae9d5}
   Method ps_Starting: Id {f49aa15f-a31d-40aa-9018-c096f512b197}
   Method ps_StopCondition: Id {dfca2682-b6c2-4944-af0d-ff6b52fb075f}
   Method ps_Stopped: Id {49063548-37a6-4746-8b21-23b1f293887b}
   Method ps_Stopping: Id {c4e39ad5-82ab-48dc-90f5-14c5203ee078}
   Method ps_SuspendCondition: Id {564dee04-1f14-4bdd-91d5-e12c2aaebc6e}
   Method ps_Suspended: Id {b36d6a26-6e02-4b88-af0f-fc68eeaf5014}
   Method ps_Suspending: Id {fa0edeb3-d0cc-447a-a291-534ad3f21e0d}
   Method ps_Unholding: Id {9ccb2058-7ec5-40de-a704-05cef1a2a6f5}
   Method ps_Unsuspending: Id {1ba62c12-a04d-4406-b5a0-b24588aae986}
   Method runSectionTasks: Id {f3604778-6c1a-49b5-ab2a-7c72901c3175}
   Method setOrder: Id {e2776e5b-59eb-47e7-a6d5-4049b002d6f5}
   Method unload: Id {b4f68f17-1b52-41bb-b94c-6f96adbd4e44} *)
